FUNCTION F_DegPerSecToDegPerMin : LREAL
VAR_INPUT
	fValue : LREAL; // °/s value
END_VAR
VAR
END_VAR

 F_DegPerSecToDegPerMin := fValue * 60; // °/s -> °/min

END_FUNCTION

(* stored: Version 1.1.0.1, ProductVersion 3.1.4024.12
   POU F_DegPerSecToDegPerMin: Id {ab048381-f416-4079-a6f8-e671d40f6bef}, SpecialFunc None *)
